// TIA Portal V20 export
TYPE "ROUT_Conf_Bucle_Lect_SCR"
   STRUCT
      Modelo : UInt := 5;   // (0) DL PB (1) SICK PB (2) SICK_A PB (5) SICK PN (6) SICK_A PN
      AddresInicial : UInt := 0;   // Direccion Entrada / Salida del Primer Nodo de la Red
      NodoInicial : UInt := 0;   // Primer Nodo de la Red (ID profinet)
      NodoFinal : UInt := 0;   // Ultimo Nodo de la Red (ID profinet)
      Numero_Red : UInt := 1;   // Número de red en la que estan los scanners
      DB_NodosPresentes : UInt := 927;   // DD de Nodos Presentes en la Red
      SCR_Actual : UInt;   // Numero de SCR actual de la Red
   END_STRUCT;
END_TYPE
